// TwinCAT 3 PLC project PLC_1
// ProgramVersion: 3.1.4024.0
// libraries:
//   Tc2_MC2, * (Beckhoff Automation GmbH)
//   Tc2_ModbusSrv, * (Beckhoff Automation GmbH)
//   Tc2_Standard, * (Beckhoff Automation GmbH)
//   Tc2_System, * (Beckhoff Automation GmbH)
//   Tc3_Module, * (Beckhoff Automation GmbH)
// project tree:
//   DUTs/ AxisStatus.TcDUT
//   / PlcTask.TcTTO, PlcTask1.TcTTO
//   POUs/ AxisControl.TcPOU, MAIN.TcPOU
// real-time tasks:
//   TASK PlcTask: cycle T#10ms, priority 12, ADS port 350
//   TASK PlcTask1: cycle T#500us, priority 4, ADS port 351
// motion (NC):
//   TASK NC-Task 1 SAF: cycle T#500us, priority 6, ADS port 501
//   TASK NC-Task 1 SVB: cycle T#2ms, priority 8, ADS port 511
//   AXIS Axis 1 (id 1)
//     General: UnitName=°, UnitFlags=#x00000004
//     OtherSettings: AllowMotionCmdToSlave=true
//     encoder EncType=1
//     drive DrvType=5
//       Analog: TorqueSetpointScale=10, ScaleFactorActTorque=0.1
//       TimeComp: TaskDelayCycles=1
//     controller CtrType=1
//       CtrPara: PriorControlFactor=1
//         Observer: BandWidth=20
//   AXIS Axis 2 (id 2)
//     General: UnitName=°, UnitFlags=#x00000004
//     OtherSettings: AllowMotionCmdToSlave=true
//     encoder EncType=1
//     drive DrvType=5
//       Analog: TorqueSetpointScale=10, ScaleFactorActTorque=0.1
//       TimeComp: TaskDelayCycles=1
//     controller CtrType=1
//       CtrPara: PriorControlFactor=1
//         Observer: BandWidth=20
//   AXIS Axis 3 (id 3)
//     General: UnitName=°, UnitFlags=#x00000004
//     OtherSettings: AllowMotionCmdToSlave=true
//     encoder EncType=1
//     drive DrvType=5
//       Analog: TorqueSetpointScale=10, ScaleFactorActTorque=0.1
//       TimeComp: TaskDelayCycles=1
//     controller CtrType=1
//       CtrPara: PriorControlFactor=1
//         Observer: BandWidth=20
// variable links:
//   PLC 1/PLC 1 Instance <-> NC-Task 1 SAF/Axes/Axis 1
//     PlcTask1 Inputs/MAIN.Control._Axis[1].NcToPlc <-> Outputs/ToPlc
//     PlcTask1 Outputs/MAIN.Control._Axis[1].PlcToNc <-> Inputs/FromPlc
//   PLC 1/PLC 1 Instance <-> NC-Task 1 SAF/Axes/Axis 2
//     PlcTask1 Inputs/MAIN.Control._Axis[2].NcToPlc <-> Outputs/ToPlc
//     PlcTask1 Outputs/MAIN.Control._Axis[2].PlcToNc <-> Inputs/FromPlc
//   PLC 1/PLC 1 Instance <-> NC-Task 1 SAF/Axes/Axis 3
//     PlcTask1 Inputs/MAIN.Control._Axis[3].NcToPlc <-> Outputs/ToPlc
//     PlcTask1 Outputs/MAIN.Control._Axis[3].PlcToNc <-> Inputs/FromPlc

CONFIGURATION PLC_1
    RESOURCE PLC ON TwinCAT3
        TASK PlcTask(INTERVAL := T#10ms, PRIORITY := 12);
        TASK PlcTask1(INTERVAL := T#500us, PRIORITY := 4);
        PROGRAM MAIN WITH PlcTask1 : MAIN;
    END_RESOURCE
END_CONFIGURATION

// ---- DUTs/AxisStatus.TcDUT
TYPE AxisStatus :
STRUCT
	
	_Error				: BOOL;
	_ErrorID			: UDINT;
	_ErrorStop			: BOOL;
	_Disabled			: BOOL;
	_Stopping			: BOOL;
	_StandStill			: BOOL;
	_DiscreteMotion		: BOOL;
	_ContinuousMotion	: BOOL;
	_SynchronizedMotion	: BOOL;
	_Homing				: BOOL;
	_ConstantVelocity	: BOOL;
	_Accelerating		: BOOL;
	_Decelerating		: BOOL;
	_Status				: ST_AxisStatus;
	
END_STRUCT
END_TYPE

// ---- POUs/MAIN.TcPOU
PROGRAM MAIN
VAR

	Control		: AxisControl;	
	State		: BYTE;
	Positions	: ARRAY [1..3] OF LREAL;

END_VAR


// Implement AxisControl

Control.CyclicUpdate();

Control.AutoErrorCheckAndReset(AxisID := 2);

CASE State OF
	
	0:
		State := 1;
	
	1:
		IF Control.PowerOn(AxisID := 2, Override := 100) THEN
			State := 2;
		END_IF
	
	2:
		Control.MoveAtVelocity(AxisID := 2, Velocity := 90, Direction := MC_Positive_Direction);
		

END_CASE

Positions := Control.CurrentPositionModulo;

END_PROGRAM

// ---- POUs/AxisControl.TcPOU
FUNCTION_BLOCK AxisControl
VAR
	
	// Axis Reference
	_Axis					: ARRAY [1.._NumberOfAxes] OF AXIS_REF;		
	
	// Internal Variables
	_i						: UINT := 0;
	_InputToggle			: BOOL := FALSE;
	_LocalState				: UINT := 0;
	_InternalCounter		: UDINT := 0;
	_InternalCounterMax		: UDINT := 1000;
	_ErrorIDPrevious		: ARRAY [1.._NumberOfAxes] OF UDINT;
	_ErrorCount				: ARRAY [1.._NumberOfAxes] OF UINT;
	_BusyMoving				: ARRAY [1.._NumberOfAxes] OF BOOL;
	_BusyStopping			: ARRAY [1.._NumberOfAxes] OF BOOL;
	_CommandDone			: BOOL := FALSE;
	_CurrentPosition		: ARRAY [1.._NumberOfAxes] OF LREAL;
	_CurrentPositionModulo	: ARRAY [1.._NumberOfAxes] OF LREAL;
	
	// Internal Functions
	_ErrorCountTrigger		: R_TRIG;
	_DelayTimer				: TON;	
	
	// Axis States (STRUCTURE Declaration)
	_Status					: ARRAY [1.._NumberOfAxes] OF AxisStatus;
	
	// Motion Functions Blocks
	_Enable					: ARRAY [1.._NumberOfAxes] OF MC_Power;
	_Reset					: ARRAY [1.._NumberOfAxes] OF MC_Reset;
	_ReadStatus				: ARRAY [1.._NumberOfAxes] OF MC_ReadStatus;
	_WriteParameter			: MC_WriteParameter;	
	_MoveAbs1				: MC_MoveAbsolute;
	_MoveAbs2				: MC_MoveAbsolute;
	_MoveRel1				: MC_MoveRelative;
	_MoveRel2				: MC_MoveRelative;
	_MoveVel1				: MC_MoveVelocity;
	_MoveVel2				: MC_MoveVelocity;
	_StopWeak				: MC_Halt;
	_StopStrong				: MC_Stop;
		
END_VAR
VAR CONSTANT
	
	_NumberOfAxes			: UINT := 3;

END_VAR

METHOD AutoErrorCheckAndReset : BOOL
VAR_INPUT
	AxisID			: UINT;	
END_VAR

// Automatically check for errors on the NC axis, then reset them
// Use with caution, this could cause damage to a physical system if implemented without care

_ReadStatus[AxisID](Axis := _Axis[AxisID]);
_Reset[AxisID](Axis := _Axis[AxisID]);
_ErrorCountTrigger(CLK := _Status[AxisID]._Error);

IF _ErrorCountTrigger.Q THEN
	_ErrorCount[AxisID] := _ErrorCount[AxisID] + 1;
END_IF

IF _Status[AxisID]._Error THEN
	_LocalState := 0;
	_Reset[AxisID].Execute := TRUE;
	IF _Reset[AxisID].Done THEN
		_Reset[AxisID].Execute := FALSE;
		AutoErrorCheckAndReset := TRUE;
	END_IF
END_IF
END_METHOD

PROPERTY AxisStatus : ARRAY [1.._NumberOfAxes] OF AxisStatus
GET
AxisStatus := _Status;
END_GET
SET
END_SET
END_PROPERTY

METHOD CheckForErrors : BOOL
VAR_INPUT	
	AxisID			: UINT;
END_VAR

// Check for errors on the NC axis

_ReadStatus[AxisID](Axis := _Axis[AxisID]);
_ErrorCountTrigger(CLK := _Status[AxisID]._Error);

IF _ErrorCountTrigger.Q THEN
	_ErrorCount[AxisID] := _ErrorCount[AxisID] + 1;
END_IF

IF _Status[AxisID]._Error THEN
	_LocalState := 0;
	CheckForErrors := TRUE;
END_IF
END_METHOD

PROPERTY CurrentPosition : ARRAY [1.._NumberOfAxes] OF LREAL
GET
CurrentPosition := _CurrentPosition;
END_GET
SET
END_SET
END_PROPERTY

PROPERTY CurrentPositionModulo : ARRAY [1.._NumberOfAxes] OF LREAL
GET
CurrentPositionModulo := _CurrentPositionModulo;
END_GET
SET
END_SET
END_PROPERTY

METHOD CyclicUpdate : BOOL
VAR_INPUT
END_VAR

// Update method needs to be called cyclically

_InputToggle := NOT(_InputToggle);

FOR _i := 1 TO _NumberOfAxes DO
	
	_Enable[_i]		(Axis := _Axis[_i]);
	_Reset[_i]		(Axis := _Axis[_i]);
	
	_ReadStatus[_i]
	(
		Axis 					:= _Axis[_i],
		Enable 					:= TRUE,
		Error 					=> _Status[_i]._Error,
		ErrorID 				=> _Status[_i]._ErrorID,
		ErrorStop 				=> _Status[_i]._ErrorStop,
		Disabled 				=> _Status[_i]._Disabled,
		Stopping 				=> _Status[_i]._Stopping,
		StandStill 				=> _Status[_i]._StandStill,
		DiscreteMotion 			=> _Status[_i]._DiscreteMotion,
		ContinuousMotion 		=> _Status[_i]._ContinuousMotion,
		SynchronizedMotion	 	=> _Status[_i]._SynchronizedMotion,
		Homing 					=> _Status[_i]._Homing,
		ConstantVelocity		=> _Status[_i]._ConstantVelocity,
		Accelerating 			=> _Status[_i]._Accelerating,
		Decelerating 			=> _Status[_i]._Decelerating,
		Status 					=> _Status[_i]._Status
	);
	
	_BusyMoving[_i] :=
	(
		_ReadStatus[_i].DiscreteMotion OR
		_ReadStatus[_i].ConstantVelocity OR
		_ReadStatus[_i].SynchronizedMotion
	);
	
	_BusyStopping[_i] :=
	(
		_ReadStatus[_i].Stopping
	);
	
	IF _Status[_i]._ErrorID <> 0 THEN
		_ErrorIDPrevious[_i] := _Status[_i]._ErrorID;
	END_IF
			
	_CurrentPosition[_i] := _Axis[_i].NcToPlc.ActPos;
	_CurrentPositionModulo[_i] := _Axis[_i].NcToPlc.ModuloActPos;
	
END_FOR

CyclicUpdate := TRUE;
END_METHOD

PROPERTY ErrorCount : ARRAY [1.._NumberOfAxes] OF UINT
GET
ErrorCount := _ErrorCount;
END_GET
SET
END_SET
END_PROPERTY

METHOD Halt : BOOL
VAR_INPUT
	AxisID			: UINT;
END_VAR

// Halts the axis, NOT locking the axis from further commands during its process

_StopWeak(Axis := _Axis[AxisID]);

_StopWeak.Execute			:= TRUE;

IF _StopWeak.Done THEN
	_StopWeak.Execute := FALSE;
	Halt := TRUE;
END_IF

IF _StopWeak.Error THEN
	_StopWeak.Execute := FALSE;
END_IF
END_METHOD

METHOD MoveAtVelocity : BOOL
VAR_INPUT
	AxisID			: UINT;
	Velocity		: LREAL;
	Direction		: MC_Direction;
END_VAR

// Move at a given speed in a defined direction until a stop command is activated

_MoveVel1(Axis := _Axis[AxisID]);

_MoveVel1.Velocity 			:= Velocity;
_MoveVel1.Direction			:= Direction;
_MoveVel1.Execute			:= TRUE;

IF _BusyMoving[AxisID] THEN
	_MoveVel1.Execute := FALSE;
	MoveAtVelocity := TRUE;
END_IF

IF _MoveVel1.Error THEN
	_MoveVel1.Execute := FALSE;
	MoveAtVelocity := FALSE;
END_IF
END_METHOD

METHOD MoveToPosition : BOOL
VAR_INPUT
	AxisID			: UINT;
	Position		: LREAL;
	Velocity		: LREAL;
END_VAR

// Move to a specific location at a given speed

_MoveAbs1(Axis := _Axis[AxisID]);

_MoveAbs1.Position			:= Position;
_MoveAbs1.Velocity 			:= Velocity;
_MoveAbs1.Execute			:= TRUE;

IF _MoveAbs1.Done THEN
	_MoveAbs1.Execute := FALSE;
	MoveToPosition := TRUE;
END_IF

IF _MoveAbs1.Error THEN
	_MoveAbs1.Execute := FALSE;
END_IF
END_METHOD

METHOD PowerOff : BOOL
VAR_INPUT
	Override	 	: LREAL;
	AxisID			: UINT;
END_VAR

// Disable the axis

IF Override < 0 THEN
	Override := 0;
ELSIF Override > 100 THEN
	Override := 100;	
END_IF

IF AxisID < 1 THEN
	AxisID := 1;
ELSIF AxisID > _NumberOfAxes THEN
	AxisID := 1;	
END_IF

_Enable[AxisID](Axis := _Axis[AxisID]);

_Enable[AxisID].Enable 				:= FALSE;
_Enable[AxisID].Enable_Negative 	:= FALSE;
_Enable[AxisID].Enable_Positive 	:= FALSE;
_Enable[AxisID].Override 			:= 0;

IF NOT(_Enable[AxisID].Status) THEN
	PowerOff := TRUE;
ELSIF _Enable[AxisID].Error THEN
	PowerOff := FALSE;
	_Enable[AxisID].Enable := FALSE;
END_IF
END_METHOD

METHOD PowerOffAll : BOOL
VAR_INPUT
END_VAR

// Enable all axes

FOR _i := 1 TO _NumberOfAxes BY 1 DO
	_Enable[_i](Axis := _Axis[_i]);
END_FOR

CASE _LocalState OF 
	
	0:
		_LocalState := 1;
	
	1:
		FOR _i := 1 TO _NumberOfAxes BY 1 DO
			_Enable[_i](Axis := _Axis[_i]);
			_Enable[_i].Enable := FALSE;
			_Enable[_i].Enable_Negative := FALSE;
			_Enable[_i].Enable_Positive := FALSE;
			_Enable[_i].Override := 0;
		END_FOR
		_LocalState := 2;
		
	2:
		_CommandDone := TRUE;
		FOR _i := 1 TO _NumberOfAxes BY 1 DO
			IF _Enable[_i].Status THEN
				_CommandDone := FALSE;
				_InternalCounter := _InternalCounter + 1;
			END_IF
		END_FOR
		
		IF _InternalCounter >= _InternalCounterMax THEN
			_InternalCounter := 0;
			_LocalState := 0;
			PowerOffAll := FALSE;
		END_IF
		
		IF _CommandDone THEN
			_InternalCounter := 0;
			_LocalState := 3;
		END_IF
		
	3:
		_LocalState := 0;
		PowerOffAll := TRUE;

END_CASE
END_METHOD

METHOD PowerOn : BOOL
VAR_INPUT
	Override	 	: LREAL;
	AxisID			: UINT;
END_VAR

// Enable the axis

IF Override < 0 THEN
	Override := 0;
ELSIF Override > 100 THEN
	Override := 100;	
END_IF

IF AxisID < 1 THEN
	AxisID := 1;
ELSIF AxisID > _NumberOfAxes THEN
	AxisID := 1;	
END_IF

_Enable[AxisID](Axis := _Axis[AxisID]);

_Enable[AxisID].Enable 				:= TRUE;
_Enable[AxisID].Enable_Negative 	:= TRUE;
_Enable[AxisID].Enable_Positive 	:= TRUE;
_Enable[AxisID].Override 			:= 100;

IF _Enable[AxisID].Status THEN
	PowerOn := TRUE;
ELSIF _Enable[AxisID].Error THEN
	PowerOn := FALSE;
	_Enable[AxisID].Enable := FALSE;
END_IF
END_METHOD

METHOD PowerOnAll : BOOL
VAR_INPUT
	Override		: LREAL;
END_VAR

// Enable all axes

IF Override < 0 THEN
	Override := 0;
ELSIF Override > 100 THEN
	Override := 100;	
END_IF

FOR _i := 1 TO _NumberOfAxes BY 1 DO
	_Enable[_i](Axis := _Axis[_i]);
END_FOR

CASE _LocalState OF 
	
	0:
		_LocalState := 1;
	
	1:
		FOR _i := 1 TO _NumberOfAxes BY 1 DO
			_Enable[_i](Axis := _Axis[_i]);
			_Enable[_i].Enable := TRUE;
			_Enable[_i].Enable_Negative := TRUE;
			_Enable[_i].Enable_Positive := TRUE;
			_Enable[_i].Override := Override;
		END_FOR
		_LocalState := 2;
		
	2:
		_CommandDone := TRUE;
		FOR _i := 1 TO _NumberOfAxes BY 1 DO
			IF NOT(_Enable[_i].Status) THEN
				_CommandDone := FALSE;
				_InternalCounter := _InternalCounter + 1;
			END_IF
		END_FOR
		
		IF _InternalCounter >= _InternalCounterMax THEN
			_InternalCounter := 0;
			_LocalState := 0;
			PowerOnAll := FALSE;
		END_IF
		
		IF _CommandDone THEN
			_InternalCounter := 0;
			_LocalState := 3;
		END_IF
		
	3:
		_LocalState := 0;
		PowerOnAll := TRUE;

END_CASE
END_METHOD

METHOD Reset : BOOL
VAR_INPUT
	AxisID			: UINT;
END_VAR

// Reset errors on the NC axis

IF AxisID < 1 THEN
	AxisID := 1;
ELSIF AxisID > _NumberOfAxes THEN
	AxisID := 1;	
END_IF

_Reset[AxisID](Axis := _Axis[AxisID]);

_Reset[AxisID].Execute 			:= TRUE;

IF _Reset[AxisID].Done THEN
	_Reset[AxisID].Execute := FALSE;
	Reset := TRUE;
END_IF
END_METHOD

METHOD ReversingSequence : BOOL
VAR_INPUT
	AxisID			: UINT;
	Position1				: LREAL;
	Position2				: LREAL;
	Velocity				: LREAL;
	DelayBetweenMoves		: TIME;
END_VAR

// Move to Position1, then to Position2, at a set speed with a delay between the movements

_MoveAbs1(Axis := _Axis[AxisID]);
_MoveAbs2(Axis := _Axis[AxisID]);
_DelayTimer(PT := DelayBetweenMoves);

_MoveAbs1.Position			:= Position1;
_MoveAbs1.Velocity 			:= Velocity;

_MoveAbs2.Position			:= Position2;
_MoveAbs2.Velocity 			:= Velocity;

CASE _LocalState OF
	
	0:
		_MoveAbs1.Execute := TRUE;
		IF _MoveAbs1.Done THEN
			_MoveAbs1.Execute := FALSE;
			_LocalState := 1;			
		END_IF
		
	1:
		_DelayTimer.IN := TRUE;
		IF _DelayTimer.Q THEN
			_DelayTimer.IN := FALSE;
			_LocalState := 2;
		END_IF
		
	2:
		_MoveAbs2.Execute := TRUE;
		IF _MoveAbs2.Done THEN
			_MoveAbs2.Execute := FALSE;
			_LocalState := 3;			
		END_IF
		
	3:
		_DelayTimer.IN := TRUE;
		IF _DelayTimer.Q THEN
			_DelayTimer.IN := FALSE;
			_LocalState := 4;
		END_IF
		
	4:
		_LocalState := 0;
		ReversingSequence := TRUE;

END_CASE

IF _MoveAbs1.Error OR _MoveAbs2.Error THEN
	_MoveAbs1.Execute := FALSE;
	_MoveAbs2.Execute := FALSE;
END_IF
END_METHOD

METHOD Stop : BOOL
VAR_INPUT
	AxisID			: UINT;
END_VAR

// Halts the axis, locking the axis from further commands during its process

_StopStrong(Axis := _Axis[AxisID]);

_StopStrong.Execute			:= TRUE;

IF _StopStrong.Done THEN
	_StopStrong.Execute := FALSE;
	Stop := TRUE;
END_IF

IF _StopStrong.Error THEN
	_StopStrong.Execute := FALSE;
END_IF
END_METHOD

METHOD WriteToParameter : BOOL
VAR_INPUT
	AxisID			: UINT;	
	Parameter		: MC_AxisParameter;
	Value			: LREAL;
END_VAR

IF AxisID < 1 THEN
	AxisID := 1;
ELSIF AxisID > _NumberOfAxes THEN
	AxisID := 1;	
END_IF

_WriteParameter(Axis := _Axis[AxisID]);

_WriteParameter.ParameterNumber := Parameter;
_WriteParameter.Value := Value;
_WriteParameter.Execute := TRUE;


IF _WriteParameter.Done THEN
	WriteToParameter := TRUE;
	_WriteParameter.Execute := FALSE;
ELSIF _WriteParameter.Error THEN
	WriteToParameter := FALSE;
	_WriteParameter.Execute := FALSE;
END_IF
END_METHOD

END_FUNCTION_BLOCK
